// TIA Portal V20 export
TYPE "LER_type_mzc_Communication"
// stored: Access Published
   STRUCT
      toLOGS : "zmc_DatatypetoLOGS";
      fromLOGS : "mzc_DatatypefromLOGS";
   END_STRUCT;
END_TYPE
